(* Logix 5000 project; controller EthernetIP_Demo_UR 1769-L16ER-BB1B rev 38.11; software revision 38.00 *)

TASK MainTask (continuous, watchdog 500 ms) : MainProgram

MODULES
   Local : 1769-L16ER-BB1B (PointIO 0, rev 38.11)
      UR_Robot : ETHERNET-MODULE (Ethernet 192.168.1.21, rev 1.1, Output RPI 10 ms)
      AENTR : 1734-AENTR (Ethernet 192.168.1.100, rev 6.12, Output RPI 20 ms)   // Extended I/O
         Light_Outputs : 1734-OB8E (PointIO 1, rev 3.22)
      Discrete_IO : Embedded (PointIO 1, rev 38.1, Output RPI 20 ms)
           Local:1:I.Data.0   // PB-1 Green
           Local:1:I.Data.1   // PB-2 Yellow
           Local:1:I.Data.2   // PB-3 Red
           Local:1:I.Data.3   // PB-4 Blue
END_MODULES

VAR_GLOBAL   (* controller tags *)
   Button_Pressed : DINT := 3;
   Candy_1_Count : DINT;
   Candy_2_Count : DINT := 1;
   Candy_3_Count : DINT;
   Candy_4_Count : DINT;
   Candy_Selected : DINT := 2;
   COUNTER_ROBOT_ACTIVE : DINT;
   Current_Light : DINT := 2;
   Disp_Light_1 : ALIAS FOR AENTR:1:O.3;
   Disp_Light_2 : ALIAS FOR AENTR:1:O.2;
   Disp_Light_3 : ALIAS FOR AENTR:1:O.1;
   Disp_Light_4 : ALIAS FOR AENTR:1:O.0;
   Game_State : DINT;
   Games_Played : DINT := 1;
   HMI_Difficulty : DINT := 3;
   HMI_Lose : BOOL;
   HMI_Restart : BOOL;
   HMI_Start : BOOL;
   HMI_StopCycle : BOOL;
   HMI_UR_Zero : BOOL;
   HMI_Win : BOOL;
   Light_Attract : BOOL;
   Light_Test : BOOL;
   OS_Button_1 : BOOL;
   OS_Button_2 : BOOL;
   OS_Button_3 : BOOL;
   OS_Button_4 : BOOL;
   OS_Button_Captured : BOOL;
   OS_Candy_Count : BOOL;
   OS_Games_Played : BOOL;
   OS_HMI_Restart : BOOL;
   OS_HMI_Start : BOOL;
   OS_Sound : BOOL;
   OS_State1_State2 : BOOL;
   OS_State2_State3 : BOOL;
   OS_UR_Done : BOOL;
   OS_UR_Start : BOOL;
   P55_RotZ : ALIAS FOR URO.Float.Registers[5];
   PB1 : ALIAS FOR Local:1:I.Data.0;
   PB2 : ALIAS FOR Local:1:I.Data.1;
   PB3 : ALIAS FOR Local:1:I.Data.2;
   PB4 : ALIAS FOR Local:1:I.Data.3;
   PL1 : ALIAS FOR Local:1:O.Data.0;   // PL-1: Green
   PL2 : ALIAS FOR Local:1:O.Data.1;   // PL-2: Yellow
   PL3 : ALIAS FOR Local:1:O.Data.2;   // PL-3: Red
   PL4 : ALIAS FOR Local:1:O.Data.3;   // PL-4: Blue
   PS5_Joint6Vel : ALIAS FOR URO.Float.Registers[6];
   PS5_Mode : DINT;
   PS5_RotX : ALIAS FOR URO.Float.Registers[3];
   PS5_RotY : ALIAS FOR URO.Float.Registers[4];
   PS5_VelX : ALIAS FOR URO.Float.Registers[0];
   PS5_VelY : ALIAS FOR URO.Float.Registers[1];
   PS5_VelZ : ALIAS FOR URO.Float.Registers[2];
   Robot_Activated : BOOL;
   SEQ_CTRL_Attract : CONTROL;
   SEQ_CTRL_Cycle : CONTROL;
   SEQ_DATA_Attract : DINT[7] := ([1] := 9, [2] := 6, [3] := 9, [4] := 6, [6] := 15);
        [0]   // Light 1
        [1]   // Light 2
        [2]   // Light 3
        [3]   // Light 4
   SEQ_DATA_Cycle : DINT[5] := ([1] := 1, [2] := 2, [3] := 4, [4] := 8);
   SEQ_DEST : DINT := 6;
   SEQ_MASK : DINT := 15;
   Sound : BOOL[32];
   Sound_Active : BOOL;
   Start_ONS : BOOL;
   temp_dint : DINT := 150;
   temp_index : DINT;
   Timer_Attract_Off : TIMER;
   Timer_Attract_On : TIMER;
   Timer_Cycle_Speed : TIMER;
   Timer_Done_Pause : TIMER;
   Timer_Fast_On : BOOL;
   Timer_Med_On : BOOL;
   TIMER_ROBOT_ACTIVE : TIMER;
   TIMER_SEQ : TIMER;
   Timer_Sound : TIMER;
   Timer_Tower_Fast : TIMER;
   Timer_Tower_Med : TIMER;
   Timer_Tower_Slow : TIMER;
   Toggle_ONS : BOOL;
   Tower_Blue : ALIAS FOR AENTR:1:O.4;
   Tower_Fast_On : BOOL;
   Tower_Green : ALIAS FOR AENTR:1:O.5;
   Tower_Med_On : BOOL;
   Tower_Red : ALIAS FOR AENTR:1:O.7;
   Tower_Slow_On : BOOL := 1;
   Tower_Yellow : ALIAS FOR AENTR:1:O.6;
   Trigger_RobotStart : BOOL;
   UR_Busy : ALIAS FOR URI.Bit.Registers[0];
   UR_ContMode : ALIAS FOR URO.Bit.Registers[1];
   UR_CurrentProg : ALIAS FOR URI.Int.Registers[0];
   UR_Done : ALIAS FOR URI.Bit.Registers[2];
   UR_EStop : ALIAS FOR URI.Safety.ES;
   UR_PowerOn : ALIAS FOR URI.Robot.PW;
   UR_ProgCmd : ALIAS FOR URO.Int.Registers[0];
   UR_ProgNum : DINT;
   UR_ProgRunning : ALIAS FOR URI.Robot.PR;
   UR_Ready : ALIAS FOR URI.Bit.Registers[1];
   UR_SafetyNormal : ALIAS FOR URI.Safety.NO;
   UR_Search : ALIAS FOR URO.Bit.Registers[3];
   UR_StartFlag : ALIAS FOR URO.Bit.Registers[0];
   URI : UR_T2O_Assembly_Combined;
   URO : UR_O2T_Assembly_Combined;
   Win_Flag : BOOL;
END_VAR

PROGRAM MainProgram   (* main routine MainRoutine *)
VAR
   alwayson : BOOL;
END_VAR

ROUTINE MainRoutine   (* ladder *)
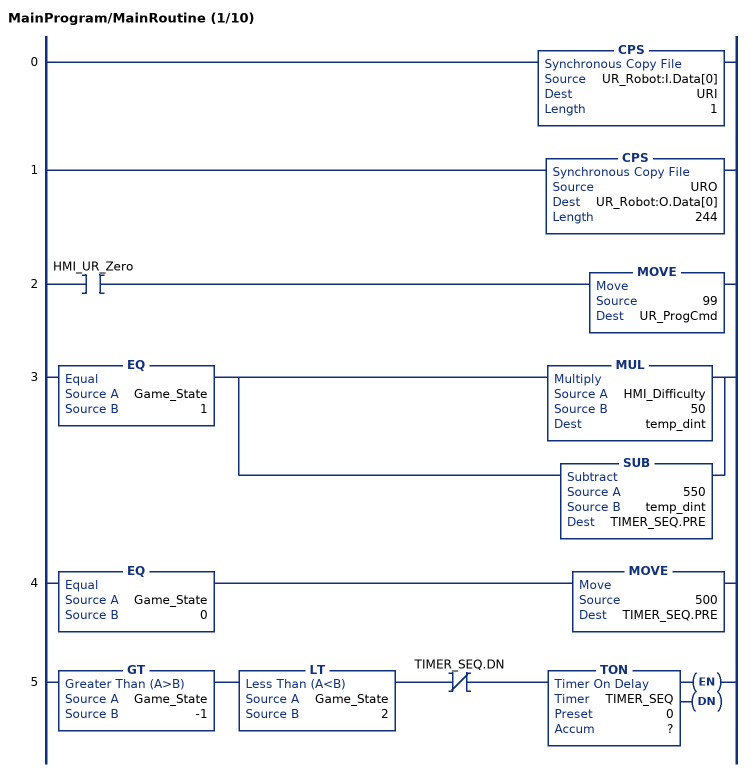
   0: CPS(UR_Robot:I.Data[0],URI,1);
   1: CPS(URO,UR_Robot:O.Data[0],244);
   2: XIC(HMI_UR_Zero)MOVE(99,UR_ProgCmd);
   3: EQ(Game_State,1)[MUL(HMI_Difficulty,50,temp_dint) ,SUB(550,temp_dint,TIMER_SEQ.PRE) ];
   4: EQ(Game_State,0)MOVE(500,TIMER_SEQ.PRE);
   5: GT(Game_State,-1)LT(Game_State,2)XIO(TIMER_SEQ.DN)TON(TIMER_SEQ,?,?);
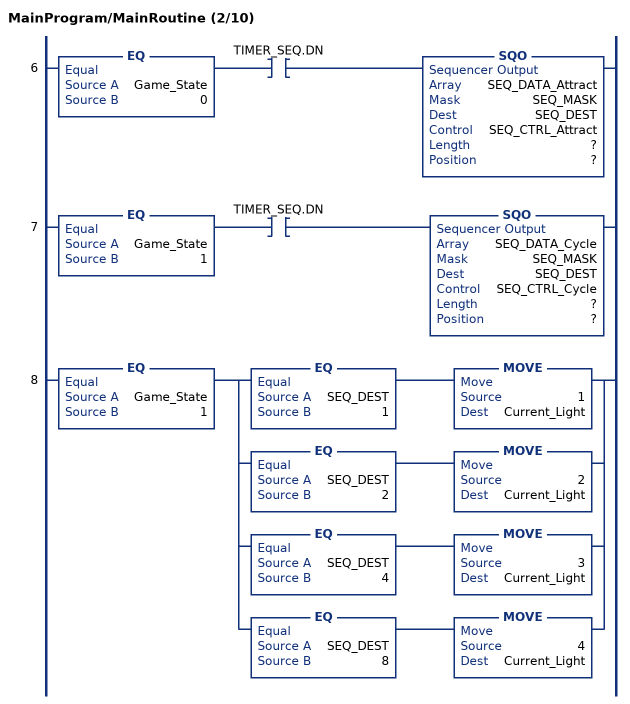
   6: EQ(Game_State,0)XIC(TIMER_SEQ.DN)SQO(SEQ_DATA_Attract,SEQ_MASK,SEQ_DEST,SEQ_CTRL_Attract,?,?);
   7: EQ(Game_State,1)XIC(TIMER_SEQ.DN)SQO(SEQ_DATA_Cycle,SEQ_MASK,SEQ_DEST,SEQ_CTRL_Cycle,?,?);
   8: EQ(Game_State,1)[EQ(SEQ_DEST,1) MOVE(1,Current_Light) ,[EQ(SEQ_DEST,2) MOVE(2,Current_Light) ,[EQ(SEQ_DEST,4) MOVE(3,Current_Light) ,EQ(SEQ_DEST,8) MOVE(4,Current_Light) ] ] ];
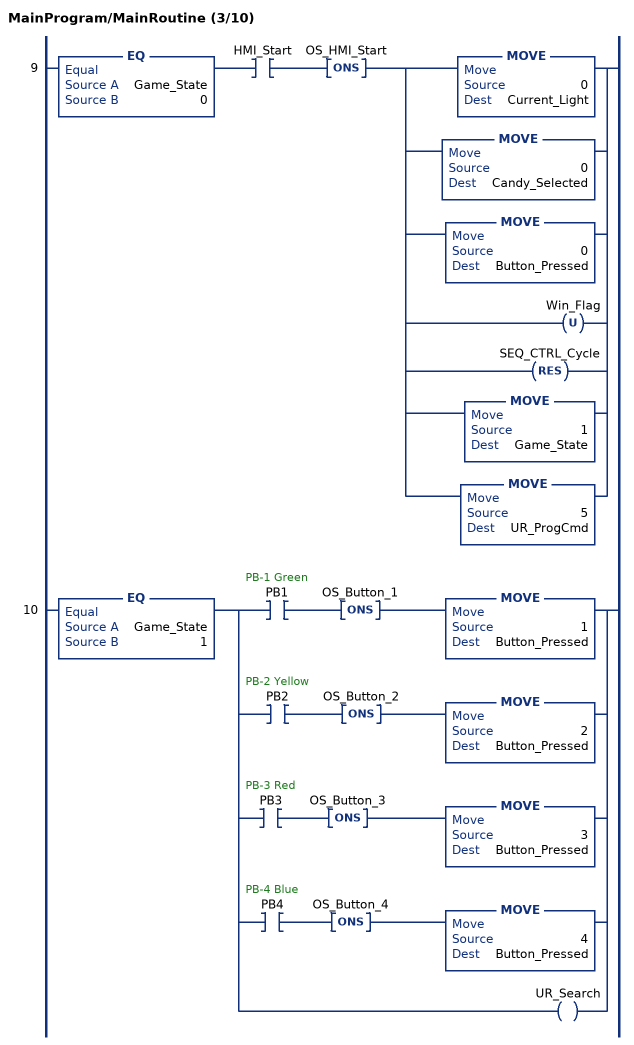
   9: EQ(Game_State,0)XIC(HMI_Start)ONS(OS_HMI_Start)[MOVE(0,Current_Light) ,[MOVE(0,Candy_Selected) ,[MOVE(0,Button_Pressed) ,[OTU(Win_Flag) ,[RES(SEQ_CTRL_Cycle) ,[MOVE(1,Game_State) ,MOVE(5,UR_ProgCmd) ] ] ] ] ] ];
   10: EQ(Game_State,1)[XIC(PB1) ONS(OS_Button_1) MOVE(1,Button_Pressed) ,[XIC(PB2) ONS(OS_Button_2) MOVE(2,Button_Pressed) ,[XIC(PB3) ONS(OS_Button_3) MOVE(3,Button_Pressed) ,[XIC(PB4) ONS(OS_Button_4) MOVE(4,Button_Pressed) ,OTE(UR_Search) ] ] ] ];
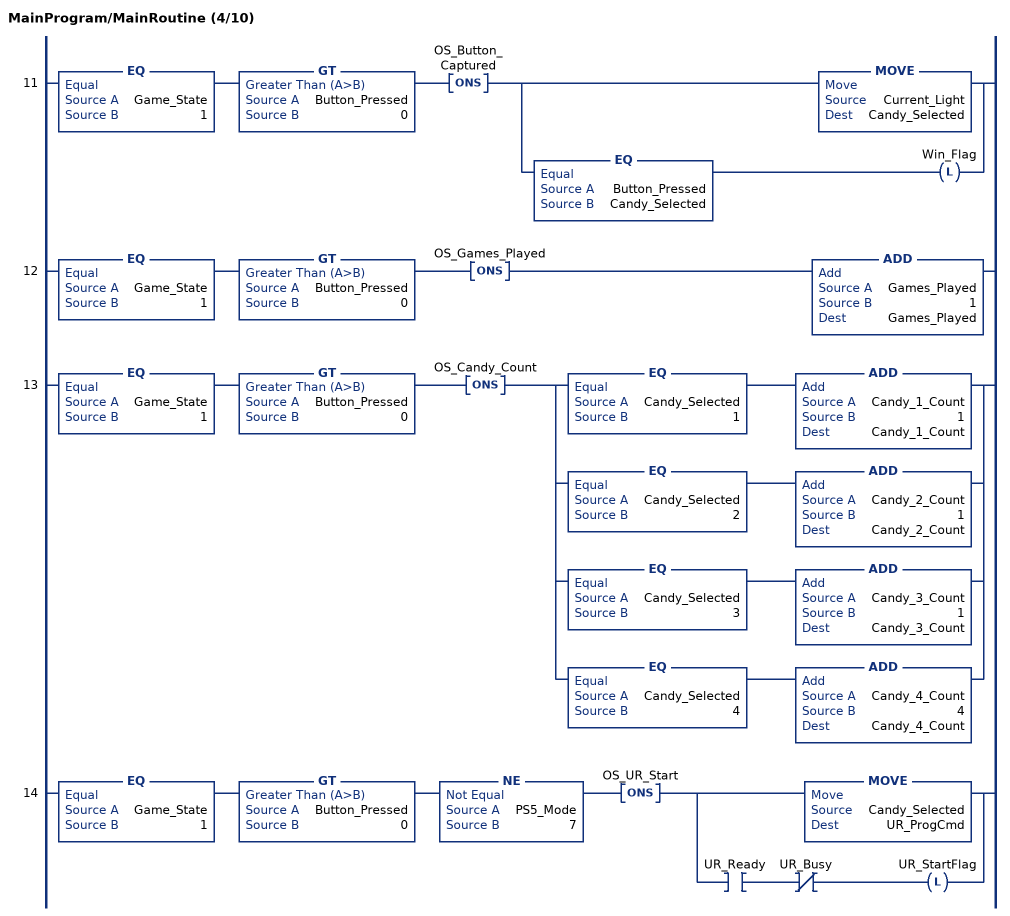
   11: EQ(Game_State,1)GT(Button_Pressed,0)ONS(OS_Button_Captured)[MOVE(Current_Light,Candy_Selected) ,EQ(Button_Pressed,Candy_Selected) OTL(Win_Flag) ];
   12: EQ(Game_State,1)GT(Button_Pressed,0)ONS(OS_Games_Played)ADD(Games_Played,1,Games_Played);
   13: EQ(Game_State,1)GT(Button_Pressed,0)ONS(OS_Candy_Count)[EQ(Candy_Selected,1) ADD(Candy_1_Count,1,Candy_1_Count) ,[EQ(Candy_Selected,2) ADD(Candy_2_Count,1,Candy_2_Count) ,[EQ(Candy_Selected,3) ADD(Candy_3_Count,1,Candy_3_Count) ,EQ(Candy_Selected,4) ADD(Candy_4_Count,4,Candy_4_Count) ] ] ];
   14: EQ(Game_State,1)GT(Button_Pressed,0)NE(PS5_Mode,7)ONS(OS_UR_Start)[MOVE(Candy_Selected,UR_ProgCmd) ,XIC(UR_Ready) XIO(UR_Busy) OTL(UR_StartFlag) ];
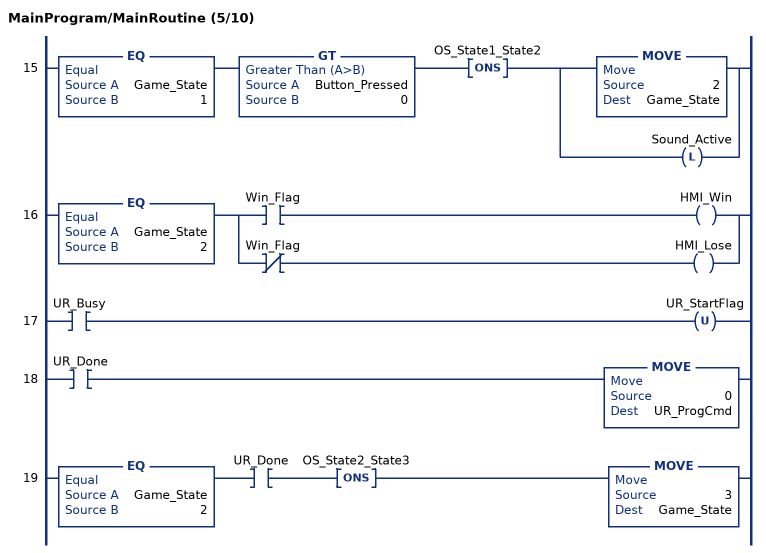
   15: EQ(Game_State,1)GT(Button_Pressed,0)ONS(OS_State1_State2)[MOVE(2,Game_State) ,OTL(Sound_Active) ];
   16: EQ(Game_State,2)[XIC(Win_Flag) OTE(HMI_Win) ,XIO(Win_Flag) OTE(HMI_Lose) ];
   17: XIC(UR_Busy)OTU(UR_StartFlag);
   18: XIC(UR_Done)MOVE(0,UR_ProgCmd);
   19: EQ(Game_State,2)XIC(UR_Done)ONS(OS_State2_State3)MOVE(3,Game_State);
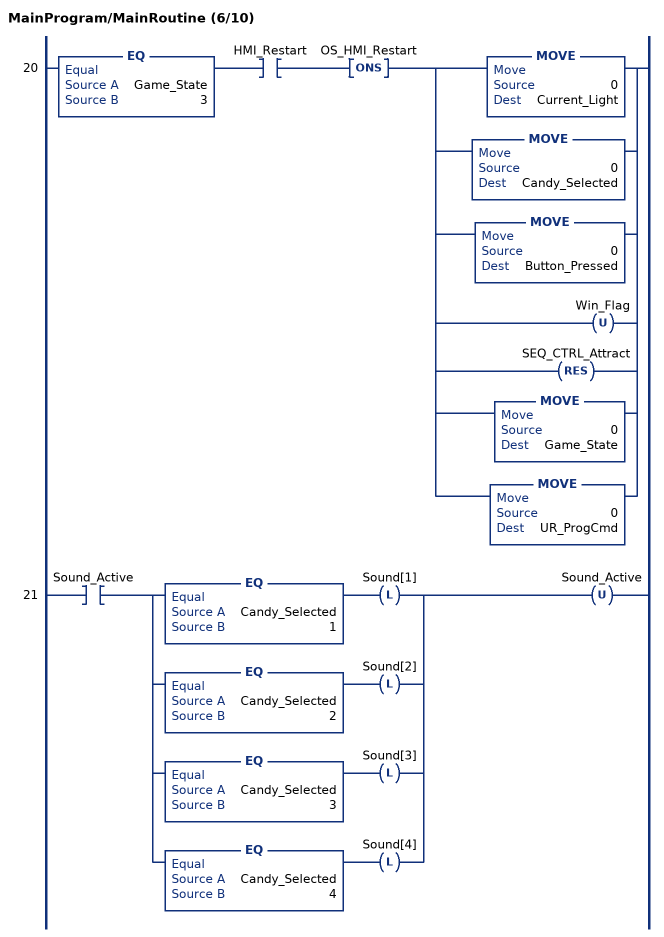
   20: EQ(Game_State,3)XIC(HMI_Restart)ONS(OS_HMI_Restart)[MOVE(0,Current_Light) ,[MOVE(0,Candy_Selected) ,[MOVE(0,Button_Pressed) ,[OTU(Win_Flag) ,[RES(SEQ_CTRL_Attract) ,[MOVE(0,Game_State) ,MOVE(0,UR_ProgCmd) ] ] ] ] ] ];
   21: XIC(Sound_Active)[EQ(Candy_Selected,1) OTL(Sound[1]) ,[EQ(Candy_Selected,2) OTL(Sound[2]) ,[EQ(Candy_Selected,3) OTL(Sound[3]) ,EQ(Candy_Selected,4) OTL(Sound[4]) ] ] ]OTU(Sound_Active);
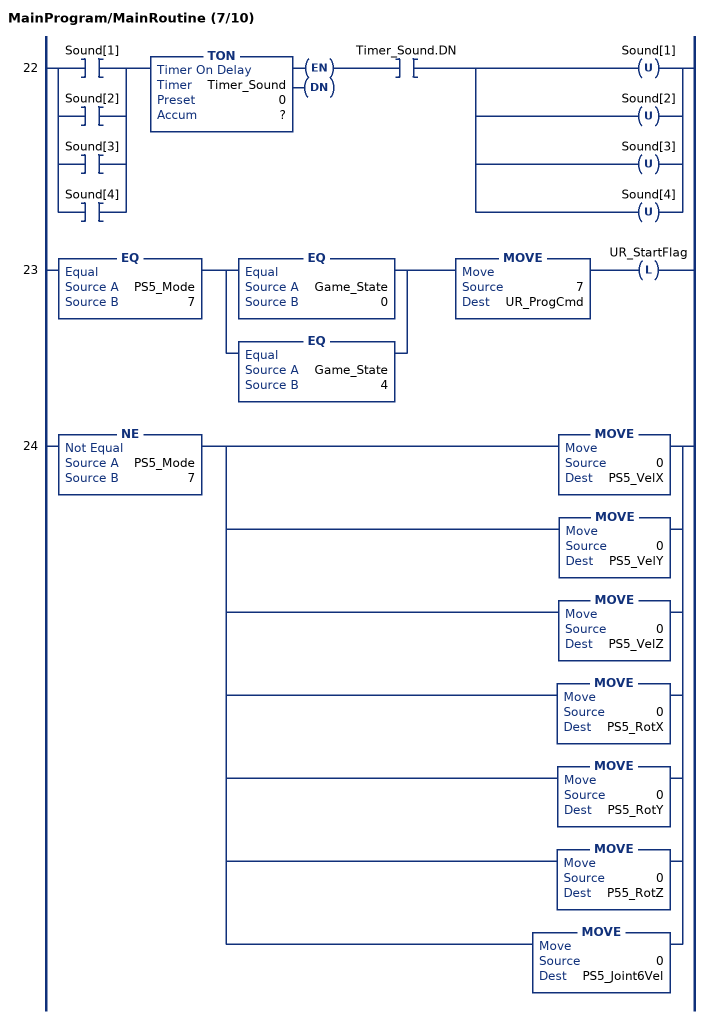
   22: [XIC(Sound[1]) ,[XIC(Sound[2]) ,[XIC(Sound[3]) ,XIC(Sound[4]) ] ] ]TON(Timer_Sound,?,?)XIC(Timer_Sound.DN)[OTU(Sound[1]) ,[OTU(Sound[2]) ,[OTU(Sound[3]) ,OTU(Sound[4]) ] ] ];
   23: EQ(PS5_Mode,7)[EQ(Game_State,0) ,EQ(Game_State,4) ]MOVE(7,UR_ProgCmd)OTL(UR_StartFlag);
   24: NE(PS5_Mode,7)[MOVE(0,PS5_VelX) ,[MOVE(0,PS5_VelY) ,[MOVE(0,PS5_VelZ) ,[MOVE(0,PS5_RotX) ,[MOVE(0,PS5_RotY) ,[MOVE(0,P55_RotZ) ,MOVE(0,PS5_Joint6Vel) ] ] ] ] ] ];
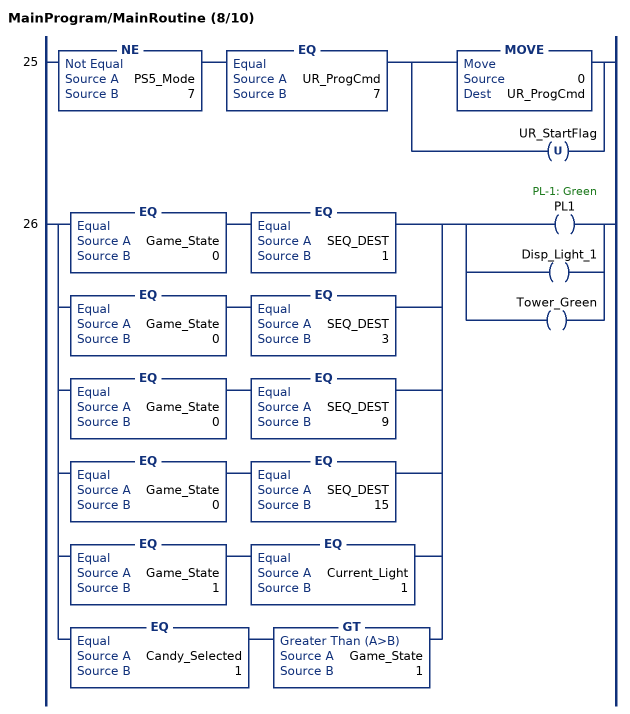
   25: NE(PS5_Mode,7)EQ(UR_ProgCmd,7)[MOVE(0,UR_ProgCmd) ,OTU(UR_StartFlag) ];
   26: [EQ(Game_State,0) EQ(SEQ_DEST,1) ,[EQ(Game_State,0) EQ(SEQ_DEST,3) ,[EQ(Game_State,0) EQ(SEQ_DEST,9) ,[EQ(Game_State,0) EQ(SEQ_DEST,15) ,[EQ(Game_State,1) EQ(Current_Light,1) ,EQ(Candy_Selected,1) GT(Game_State,1) ] ] ] ] ][OTE(PL1) ,[OTE(Disp_Light_1) ,OTE(Tower_Green) ] ];
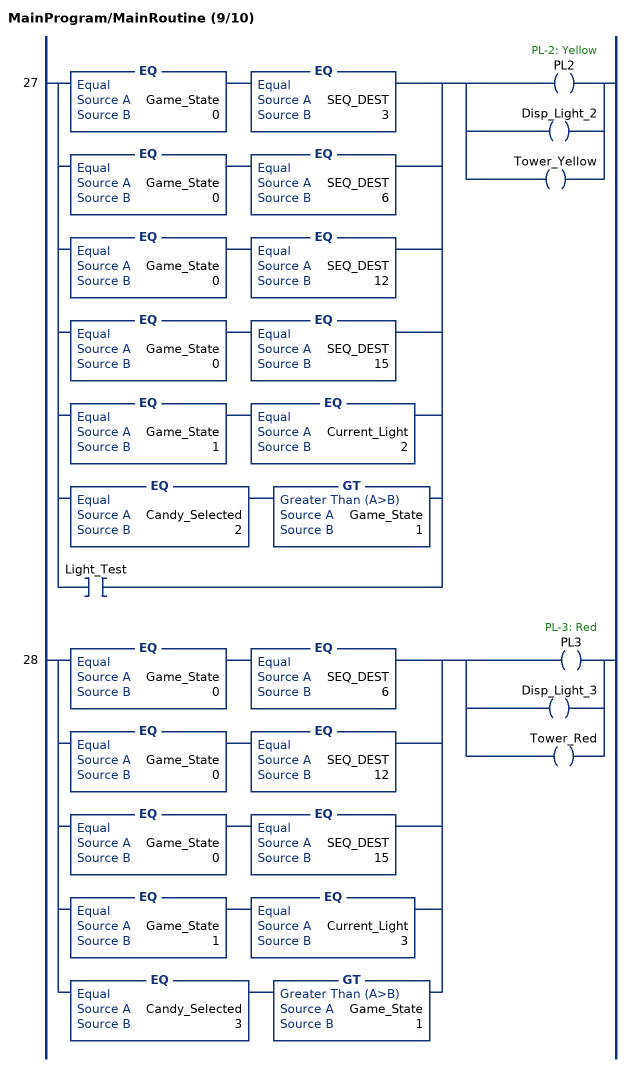
   27: [EQ(Game_State,0) EQ(SEQ_DEST,3) ,[EQ(Game_State,0) EQ(SEQ_DEST,6) ,[EQ(Game_State,0) EQ(SEQ_DEST,12) ,[EQ(Game_State,0) EQ(SEQ_DEST,15) ,[EQ(Game_State,1) EQ(Current_Light,2) ,[EQ(Candy_Selected,2) GT(Game_State,1) ,XIC(Light_Test) ] ] ] ] ] ][OTE(PL2) ,[OTE(Disp_Light_2) ,OTE(Tower_Yellow) ] ];
   28: [EQ(Game_State,0) EQ(SEQ_DEST,6) ,[EQ(Game_State,0) EQ(SEQ_DEST,12) ,[EQ(Game_State,0) EQ(SEQ_DEST,15) ,[EQ(Game_State,1) EQ(Current_Light,3) ,EQ(Candy_Selected,3) GT(Game_State,1) ] ] ] ][OTE(PL3) ,[OTE(Disp_Light_3) ,OTE(Tower_Red) ] ];
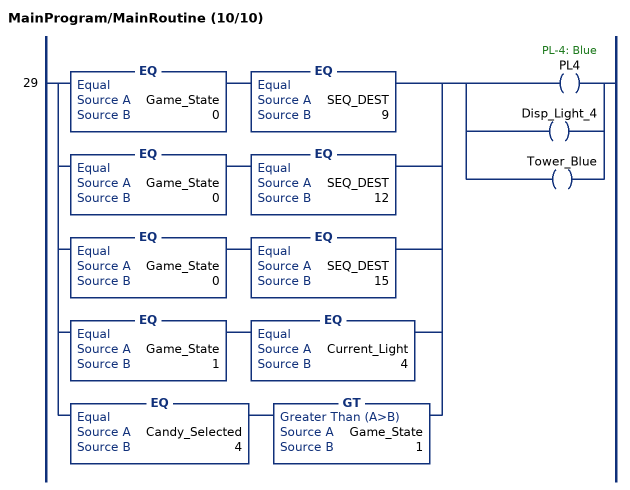
   29: [EQ(Game_State,0) EQ(SEQ_DEST,9) ,[EQ(Game_State,0) EQ(SEQ_DEST,12) ,[EQ(Game_State,0) EQ(SEQ_DEST,15) ,[EQ(Game_State,1) EQ(Current_Light,4) ,EQ(Candy_Selected,4) GT(Game_State,1) ] ] ] ][OTE(PL4) ,[OTE(Disp_Light_4) ,OTE(Tower_Blue) ] ];
END_ROUTINE
END_PROGRAM
